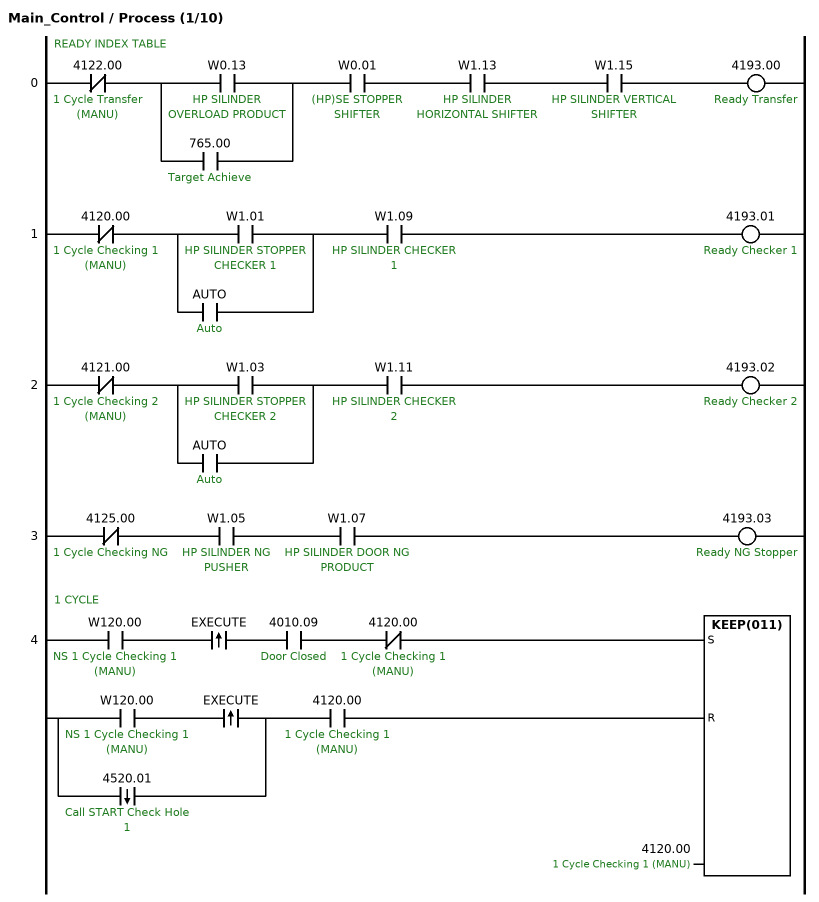
; [picture p24: Main_Control / Process, rungs 0-4]
; rung 0: READY INDEX TABLE
LDNOT 4122.00  ; 1 Cycle Transfer (MANU)
LD W0.13  ; HP SILINDER OVERLOAD PRODUCT
OR 765.00  ; Target Achieve
ANDLD
AND W0.01  ; (HP)SE STOPPER SHIFTER
AND W1.13  ; HP SILINDER HORIZONTAL SHIFTER
AND W1.15  ; HP SILINDER VERTICAL SHIFTER
OUT 4193.00  ; Ready Transfer
; rung 1
LDNOT 4120.00  ; 1 Cycle Checking 1 (MANU)
LD W1.01  ; HP SILINDER STOPPER CHECKER 1
OR AUTO  ; Auto
ANDLD
AND W1.09  ; HP SILINDER CHECKER 1
OUT 4193.01  ; Ready Checker 1
; rung 2
LDNOT 4121.00  ; 1 Cycle Checking 2 (MANU)
LD W1.03  ; HP SILINDER STOPPER CHECKER 2
OR AUTO  ; Auto
ANDLD
AND W1.11  ; HP SILINDER CHECKER 2
OUT 4193.02  ; Ready Checker 2
; rung 3
LDNOT 4125.00  ; 1 Cycle Checking NG
AND W1.05  ; HP SILINDER NG PUSHER
AND W1.07  ; HP SILINDER DOOR NG PRODUCT
OUT 4193.03  ; Ready NG Stopper
; rung 4: 1 CYCLE
LD W120.00  ; NS 1 Cycle Checking 1 (MANU)
@AND EXECUTE
AND 4010.09  ; Door Closed
ANDNOT 4120.00  ; 1 Cycle Checking 1 (MANU)
LD W120.00  ; NS 1 Cycle Checking 1 (MANU)
@AND EXECUTE
%OR 4520.01  ; Call START Check Hole 1
AND 4120.00  ; 1 Cycle Checking 1 (MANU)
KEEP(011) 4120.00  ; 1 Cycle Checking 1 (MANU)

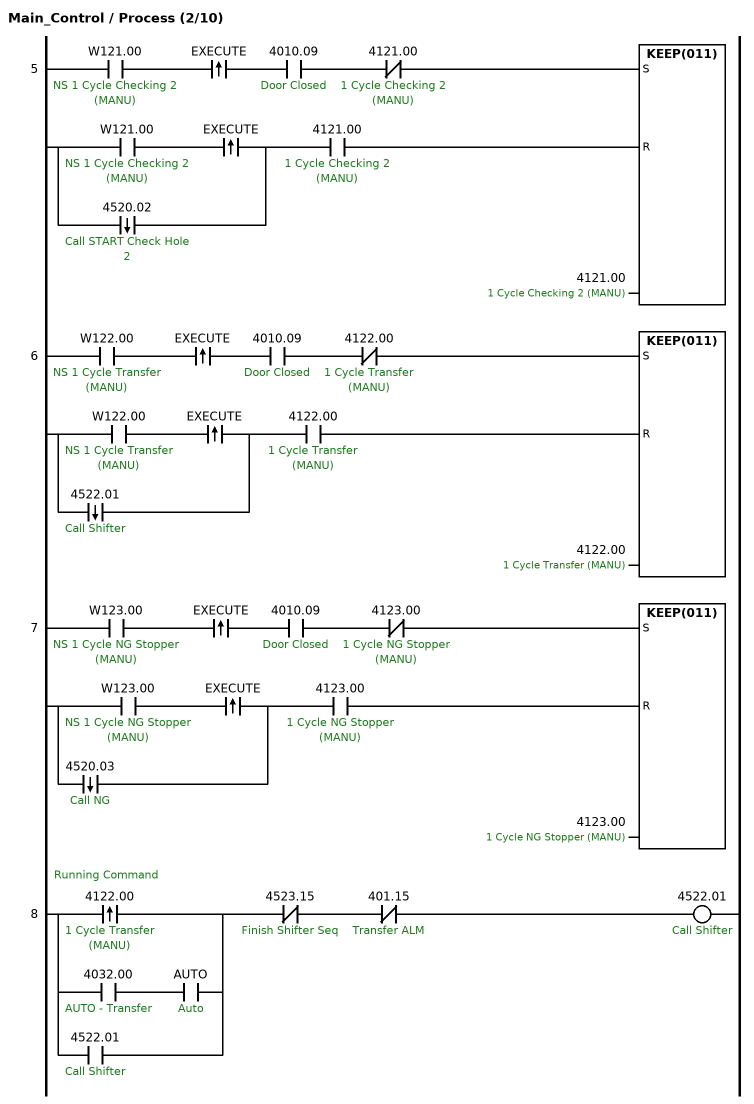
; rung 5
LD W121.00  ; NS 1 Cycle Checking 2 (MANU)
@AND EXECUTE
AND 4010.09  ; Door Closed
ANDNOT 4121.00  ; 1 Cycle Checking 2 (MANU)
LD W121.00  ; NS 1 Cycle Checking 2 (MANU)
@AND EXECUTE
%OR 4520.02  ; Call START Check Hole 2
AND 4121.00  ; 1 Cycle Checking 2 (MANU)
KEEP(011) 4121.00  ; 1 Cycle Checking 2 (MANU)
; rung 6
LD W122.00  ; NS 1 Cycle Transfer  (MANU)
@AND EXECUTE
AND 4010.09  ; Door Closed
ANDNOT 4122.00  ; 1 Cycle Transfer (MANU)
LD W122.00  ; NS 1 Cycle Transfer  (MANU)
@AND EXECUTE
%OR 4522.01  ; Call Shifter
AND 4122.00  ; 1 Cycle Transfer (MANU)
KEEP(011) 4122.00  ; 1 Cycle Transfer (MANU)
; rung 7
LD W123.00  ; NS 1 Cycle NG Stopper (MANU)
@AND EXECUTE
AND 4010.09  ; Door Closed
ANDNOT 4123.00  ; 1 Cycle NG Stopper (MANU)
LD W123.00  ; NS 1 Cycle NG Stopper (MANU)
@AND EXECUTE
%OR 4520.03  ; Call NG
AND 4123.00  ; 1 Cycle NG Stopper (MANU)
KEEP(011) 4123.00  ; 1 Cycle NG Stopper (MANU)
; rung 8: Running Command
@LD 4122.00  ; 1 Cycle Transfer (MANU)
LD 4032.00  ; AUTO - Transfer
AND AUTO  ; Auto
ORLD
OR 4522.01  ; Call Shifter
ANDNOT 4523.15  ; Finish Shifter Seq
ANDNOT 401.15  ; Transfer ALM
OUT 4522.01  ; Call Shifter

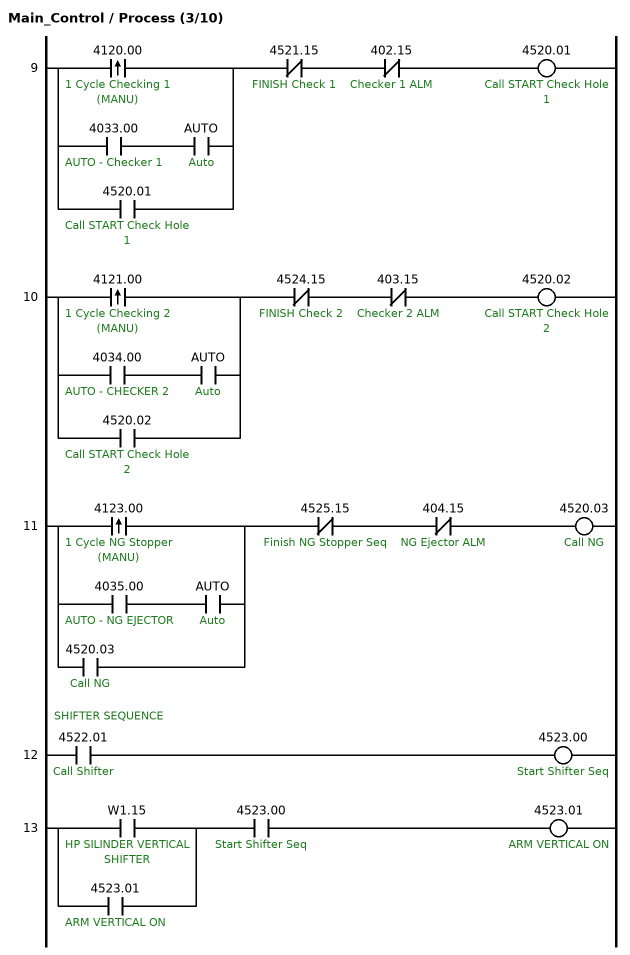
; rung 9
@LD 4120.00  ; 1 Cycle Checking 1 (MANU)
LD 4033.00  ; AUTO - Checker 1
AND AUTO  ; Auto
ORLD
OR 4520.01  ; Call START Check Hole 1
ANDNOT 4521.15  ; FINISH Check 1
ANDNOT 402.15  ; Checker 1 ALM
OUT 4520.01  ; Call START Check Hole 1
; rung 10
@LD 4121.00  ; 1 Cycle Checking 2 (MANU)
LD 4034.00  ; AUTO - CHECKER 2
AND AUTO  ; Auto
ORLD
OR 4520.02  ; Call START Check Hole 2
ANDNOT 4524.15  ; FINISH Check 2
ANDNOT 403.15  ; Checker 2 ALM
OUT 4520.02  ; Call START Check Hole 2
; rung 11
@LD 4123.00  ; 1 Cycle NG Stopper (MANU)
LD 4035.00  ; AUTO - NG EJECTOR
AND AUTO  ; Auto
ORLD
OR 4520.03  ; Call NG
ANDNOT 4525.15  ; Finish NG Stopper Seq
ANDNOT 404.15  ; NG Ejector ALM
OUT 4520.03  ; Call NG
; rung 12: SHIFTER SEQUENCE
LD 4522.01  ; Call Shifter
OUT 4523.00  ; Start Shifter Seq
; rung 13
LD W1.15  ; HP SILINDER VERTICAL SHIFTER
OR 4523.01  ; ARM VERTICAL ON
AND 4523.00  ; Start Shifter Seq
OUT 4523.01  ; ARM VERTICAL ON

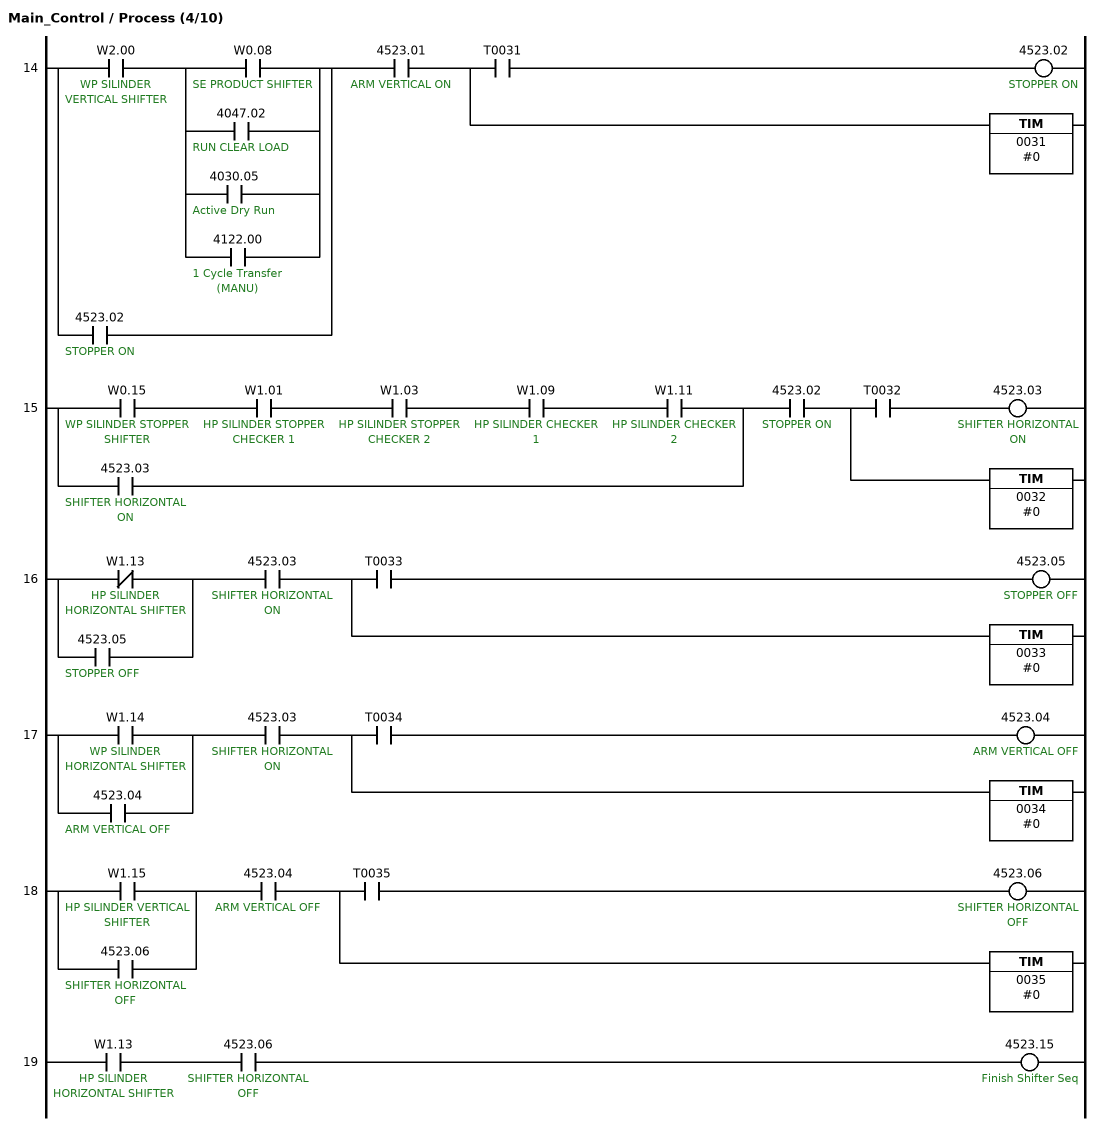
; rung 14
LD W2.00  ; WP SILINDER VERTICAL SHIFTER
LD W0.08  ; SE PRODUCT SHIFTER
OR 4047.02  ; RUN CLEAR LOAD
OR 4030.05  ; Active Dry Run
OR 4122.00  ; 1 Cycle Transfer (MANU)
ANDLD
OR 4523.02  ; STOPPER ON
AND 4523.01  ; ARM VERTICAL ON
OUT TR0
AND T0031
OUT 4523.02  ; STOPPER ON
LD TR0
TIM 0031 #0
; rung 15
LD W0.15  ; WP SILINDER STOPPER SHIFTER
AND W1.01  ; HP SILINDER STOPPER CHECKER 1
AND W1.03  ; HP SILINDER STOPPER CHECKER 2
AND W1.09  ; HP SILINDER CHECKER 1
AND W1.11  ; HP SILINDER CHECKER 2
OR 4523.03  ; SHIFTER HORIZONTAL ON
AND 4523.02  ; STOPPER ON
OUT TR0
AND T0032
OUT 4523.03  ; SHIFTER HORIZONTAL ON
LD TR0
TIM 0032 #0
; rung 16
LDNOT W1.13  ; HP SILINDER HORIZONTAL SHIFTER
OR 4523.05  ; STOPPER OFF
AND 4523.03  ; SHIFTER HORIZONTAL ON
OUT TR0
AND T0033
OUT 4523.05  ; STOPPER OFF
LD TR0
TIM 0033 #0
; rung 17
LD W1.14  ; WP SILINDER HORIZONTAL SHIFTER
OR 4523.04  ; ARM VERTICAL OFF
AND 4523.03  ; SHIFTER HORIZONTAL ON
OUT TR0
AND T0034
OUT 4523.04  ; ARM VERTICAL OFF
LD TR0
TIM 0034 #0
; rung 18
LD W1.15  ; HP SILINDER VERTICAL SHIFTER
OR 4523.06  ; SHIFTER HORIZONTAL OFF
AND 4523.04  ; ARM VERTICAL OFF
OUT TR0
AND T0035
OUT 4523.06  ; SHIFTER HORIZONTAL OFF
LD TR0
TIM 0035 #0
; rung 19
LD W1.13  ; HP SILINDER HORIZONTAL SHIFTER
AND 4523.06  ; SHIFTER HORIZONTAL OFF
OUT 4523.15  ; Finish Shifter Seq

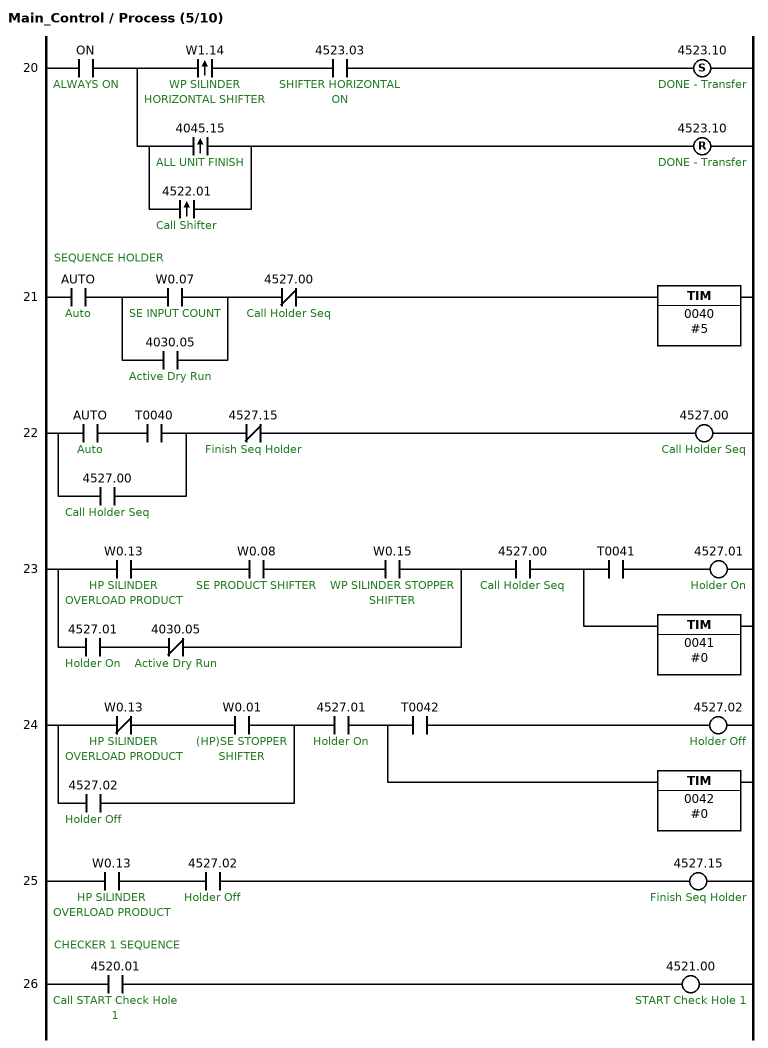
; rung 20
LD ON  ; ALWAYS ON
OUT TR0
@AND W1.14  ; WP SILINDER HORIZONTAL SHIFTER
AND 4523.03  ; SHIFTER HORIZONTAL ON
SET 4523.10  ; DONE - Transfer
LD TR0
@LD 4045.15  ; ALL UNIT FINISH
@OR 4522.01  ; Call Shifter
ANDLD
RSET 4523.10  ; DONE - Transfer
; rung 21: SEQUENCE HOLDER
LD AUTO  ; Auto
LD W0.07  ; SE INPUT COUNT
OR 4030.05  ; Active Dry Run
ANDLD
ANDNOT 4527.00  ; Call Holder Seq
TIM 0040 #5
; rung 22
LD AUTO  ; Auto
AND T0040
OR 4527.00  ; Call Holder Seq
ANDNOT 4527.15  ; Finish Seq Holder
OUT 4527.00  ; Call Holder Seq
; rung 23
LD W0.13  ; HP SILINDER OVERLOAD PRODUCT
AND W0.08  ; SE PRODUCT SHIFTER
AND W0.15  ; WP SILINDER STOPPER SHIFTER
LD 4527.01  ; Holder On
ANDNOT 4030.05  ; Active Dry Run
ORLD
AND 4527.00  ; Call Holder Seq
OUT TR0
AND T0041
OUT 4527.01  ; Holder On
LD TR0
TIM 0041 #0
; rung 24
LDNOT W0.13  ; HP SILINDER OVERLOAD PRODUCT
AND W0.01  ; (HP)SE STOPPER SHIFTER
OR 4527.02  ; Holder Off
AND 4527.01  ; Holder On
OUT TR0
AND T0042
OUT 4527.02  ; Holder Off
LD TR0
TIM 0042 #0
; rung 25
LD W0.13  ; HP SILINDER OVERLOAD PRODUCT
AND 4527.02  ; Holder Off
OUT 4527.15  ; Finish Seq Holder
; rung 26: CHECKER 1 SEQUENCE
LD 4520.01  ; Call START Check Hole 1
OUT 4521.00  ; START Check Hole 1

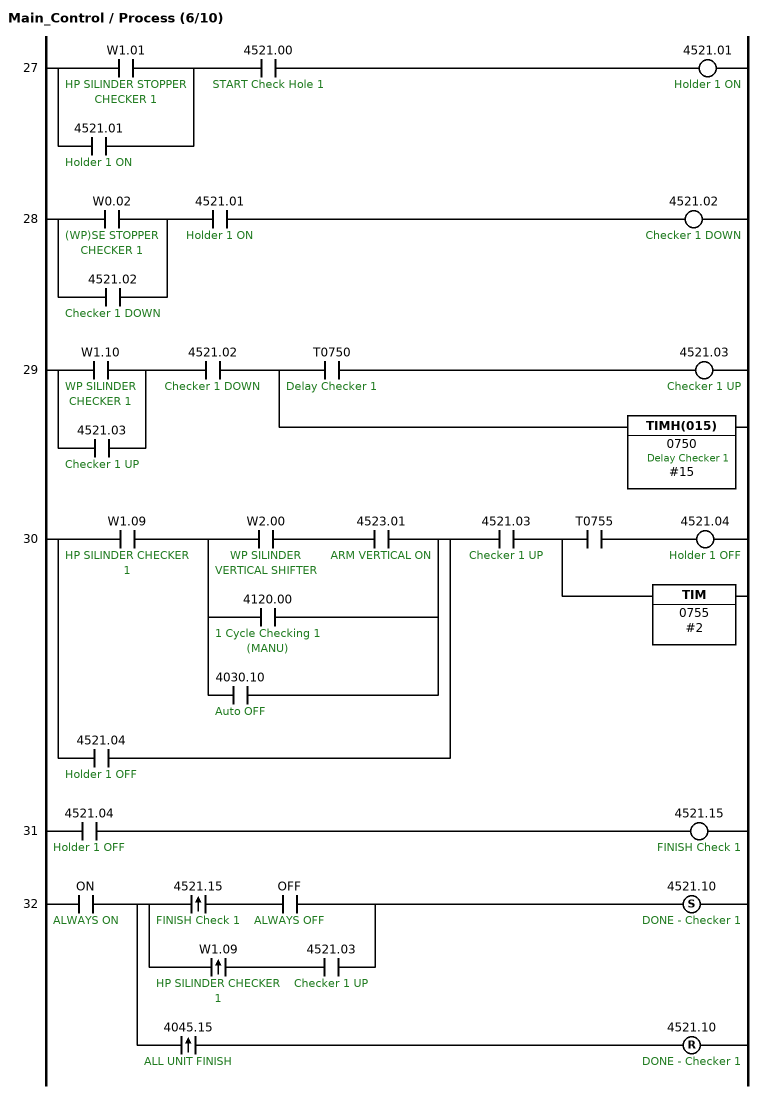
; rung 27
LD W1.01  ; HP SILINDER STOPPER CHECKER 1
OR 4521.01  ; Holder 1 ON
AND 4521.00  ; START Check Hole 1
OUT 4521.01  ; Holder 1 ON
; rung 28
LD W0.02  ; (WP)SE STOPPER CHECKER 1
OR 4521.02  ; Checker 1 DOWN
AND 4521.01  ; Holder 1 ON
OUT 4521.02  ; Checker 1 DOWN
; rung 29
LD W1.10  ; WP SILINDER CHECKER 1
OR 4521.03  ; Checker 1 UP
AND 4521.02  ; Checker 1 DOWN
OUT TR0
AND T0750  ; Delay Checker 1
OUT 4521.03  ; Checker 1 UP
LD TR0
TIMH(015) 0750 #15  ; Delay Checker 1
; rung 30
LD W1.09  ; HP SILINDER CHECKER 1
LD W2.00  ; WP SILINDER VERTICAL SHIFTER
AND 4523.01  ; ARM VERTICAL ON
OR 4120.00  ; 1 Cycle Checking 1 (MANU)
OR 4030.10  ; Auto OFF
ANDLD
OR 4521.04  ; Holder 1 OFF
AND 4521.03  ; Checker 1 UP
OUT TR0
AND T0755
OUT 4521.04  ; Holder 1 OFF
LD TR0
TIM 0755 #2
; rung 31
LD 4521.04  ; Holder 1 OFF
OUT 4521.15  ; FINISH Check 1
; rung 32
LD ON  ; ALWAYS ON
OUT TR0
@LD 4521.15  ; FINISH Check 1
AND OFF  ; ALWAYS OFF
@LD W1.09  ; HP SILINDER CHECKER 1
AND 4521.03  ; Checker 1 UP
ORLD
ANDLD
SET 4521.10  ; DONE - Checker 1
LD TR0
@AND 4045.15  ; ALL UNIT FINISH
RSET 4521.10  ; DONE - Checker 1

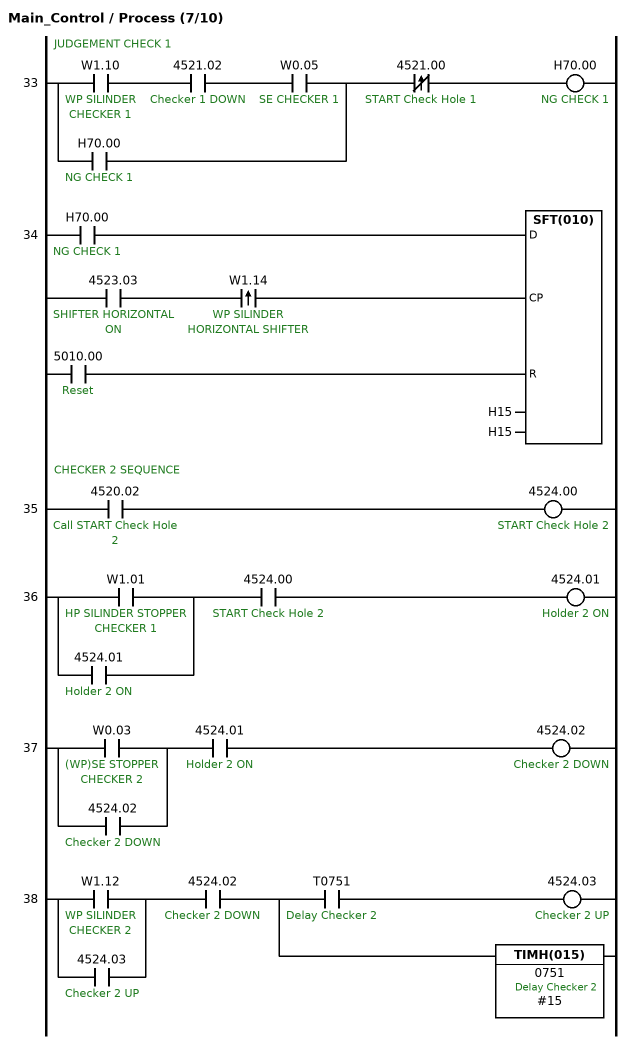
; rung 33: JUDGEMENT CHECK 1
LD W1.10  ; WP SILINDER CHECKER 1
AND 4521.02  ; Checker 1 DOWN
AND W0.05  ; SE CHECKER 1
OR H70.00  ; NG CHECK 1
@ANDNOT 4521.00  ; START Check Hole 1
OUT H70.00  ; NG CHECK 1
; rung 34
LD H70.00  ; NG CHECK 1
LD 4523.03  ; SHIFTER HORIZONTAL ON
@AND W1.14  ; WP SILINDER HORIZONTAL SHIFTER
LD 5010.00  ; Reset
SFT(010) H15 H15
; rung 35: CHECKER 2 SEQUENCE
LD 4520.02  ; Call START Check Hole 2
OUT 4524.00  ; START Check Hole 2
; rung 36
LD W1.01  ; HP SILINDER STOPPER CHECKER 1
OR 4524.01  ; Holder 2 ON
AND 4524.00  ; START Check Hole 2
OUT 4524.01  ; Holder 2 ON
; rung 37
LD W0.03  ; (WP)SE STOPPER CHECKER 2
OR 4524.02  ; Checker 2 DOWN
AND 4524.01  ; Holder 2 ON
OUT 4524.02  ; Checker 2 DOWN
; rung 38
LD W1.12  ; WP SILINDER CHECKER 2
OR 4524.03  ; Checker 2 UP
AND 4524.02  ; Checker 2 DOWN
OUT TR0
AND T0751  ; Delay Checker 2
OUT 4524.03  ; Checker 2 UP
LD TR0
TIMH(015) 0751 #15  ; Delay Checker 2

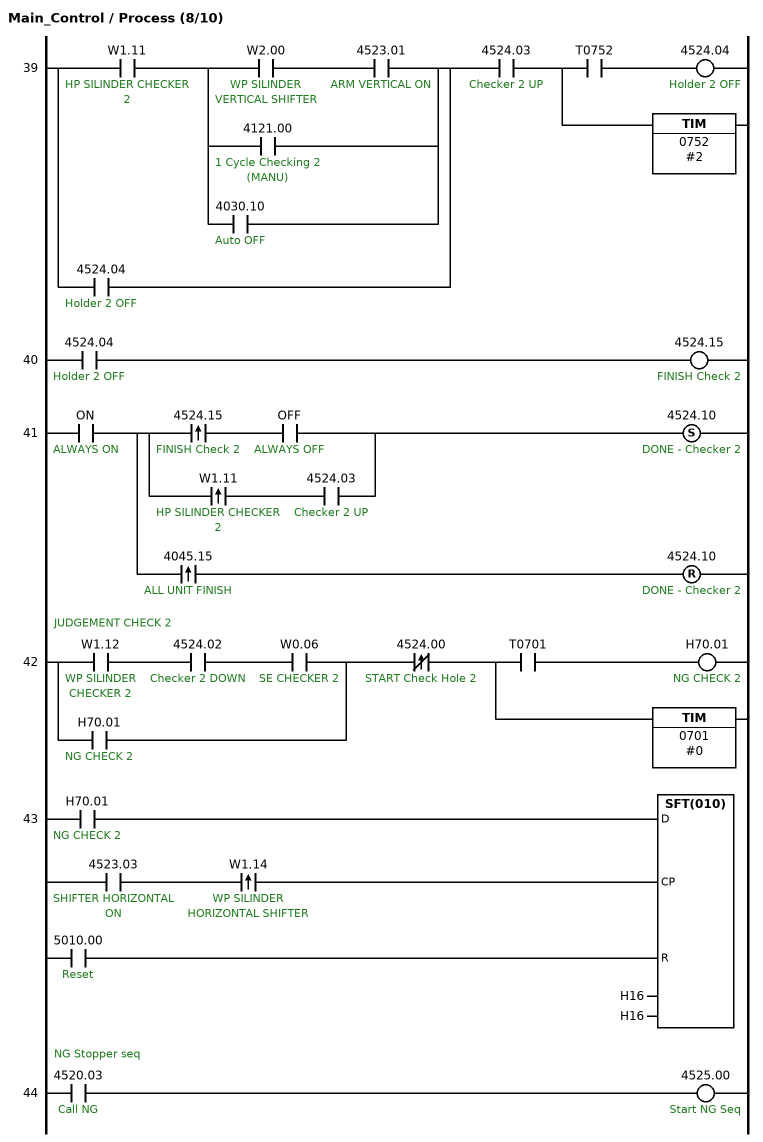
; rung 39
LD W1.11  ; HP SILINDER CHECKER 2
LD W2.00  ; WP SILINDER VERTICAL SHIFTER
AND 4523.01  ; ARM VERTICAL ON
OR 4121.00  ; 1 Cycle Checking 2 (MANU)
OR 4030.10  ; Auto OFF
ANDLD
OR 4524.04  ; Holder 2 OFF
AND 4524.03  ; Checker 2 UP
OUT TR0
AND T0752
OUT 4524.04  ; Holder 2 OFF
LD TR0
TIM 0752 #2
; rung 40
LD 4524.04  ; Holder 2 OFF
OUT 4524.15  ; FINISH Check 2
; rung 41
LD ON  ; ALWAYS ON
OUT TR0
@LD 4524.15  ; FINISH Check 2
AND OFF  ; ALWAYS OFF
@LD W1.11  ; HP SILINDER CHECKER 2
AND 4524.03  ; Checker 2 UP
ORLD
ANDLD
SET 4524.10  ; DONE - Checker 2
LD TR0
@AND 4045.15  ; ALL UNIT FINISH
RSET 4524.10  ; DONE - Checker 2
; rung 42: JUDGEMENT CHECK 2
LD W1.12  ; WP SILINDER CHECKER 2
AND 4524.02  ; Checker 2 DOWN
AND W0.06  ; SE CHECKER 2
OR H70.01  ; NG CHECK 2
@ANDNOT 4524.00  ; START Check Hole 2
OUT TR0
AND T0701
OUT H70.01  ; NG CHECK 2
LD TR0
TIM 0701 #0
; rung 43
LD H70.01  ; NG CHECK 2
LD 4523.03  ; SHIFTER HORIZONTAL ON
@AND W1.14  ; WP SILINDER HORIZONTAL SHIFTER
LD 5010.00  ; Reset
SFT(010) H16 H16
; rung 44: NG Stopper seq
LD 4520.03  ; Call NG
OUT 4525.00  ; Start NG Seq

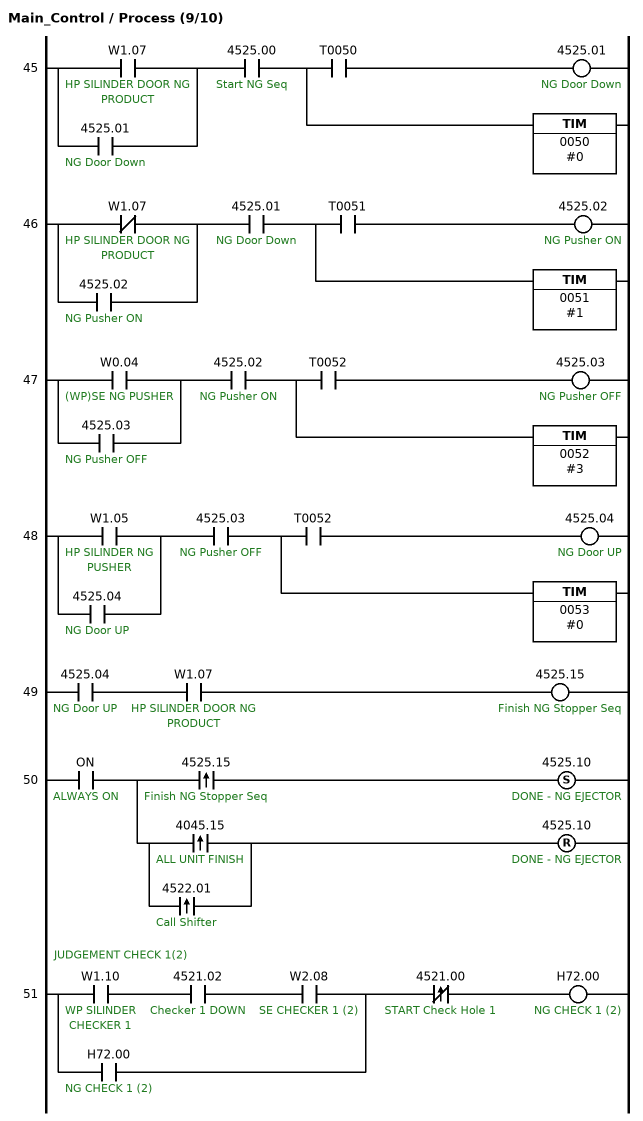
; rung 45
LD W1.07  ; HP SILINDER DOOR NG PRODUCT
OR 4525.01  ; NG Door Down
AND 4525.00  ; Start NG Seq
OUT TR0
AND T0050
OUT 4525.01  ; NG Door Down
LD TR0
TIM 0050 #0
; rung 46
LDNOT W1.07  ; HP SILINDER DOOR NG PRODUCT
OR 4525.02  ; NG Pusher ON
AND 4525.01  ; NG Door Down
OUT TR0
AND T0051
OUT 4525.02  ; NG Pusher ON
LD TR0
TIM 0051 #1
; rung 47
LD W0.04  ; (WP)SE NG PUSHER
OR 4525.03  ; NG Pusher OFF
AND 4525.02  ; NG Pusher ON
OUT TR0
AND T0052
OUT 4525.03  ; NG Pusher OFF
LD TR0
TIM 0052 #3
; rung 48
LD W1.05  ; HP SILINDER NG PUSHER
OR 4525.04  ; NG Door UP
AND 4525.03  ; NG Pusher OFF
OUT TR0
AND T0052
OUT 4525.04  ; NG Door UP
LD TR0
TIM 0053 #0
; rung 49
LD 4525.04  ; NG Door UP
AND W1.07  ; HP SILINDER DOOR NG PRODUCT
OUT 4525.15  ; Finish NG Stopper Seq
; rung 50
LD ON  ; ALWAYS ON
OUT TR0
@AND 4525.15  ; Finish NG Stopper Seq
SET 4525.10  ; DONE - NG EJECTOR
LD TR0
@LD 4045.15  ; ALL UNIT FINISH
@OR 4522.01  ; Call Shifter
ANDLD
RSET 4525.10  ; DONE - NG EJECTOR
; rung 51: JUDGEMENT CHECK 1(2)
LD W1.10  ; WP SILINDER CHECKER 1
AND 4521.02  ; Checker 1 DOWN
AND W2.08  ; SE CHECKER 1 (2)
OR H72.00  ; NG CHECK 1 (2)
@ANDNOT 4521.00  ; START Check Hole 1
OUT H72.00  ; NG CHECK 1 (2)

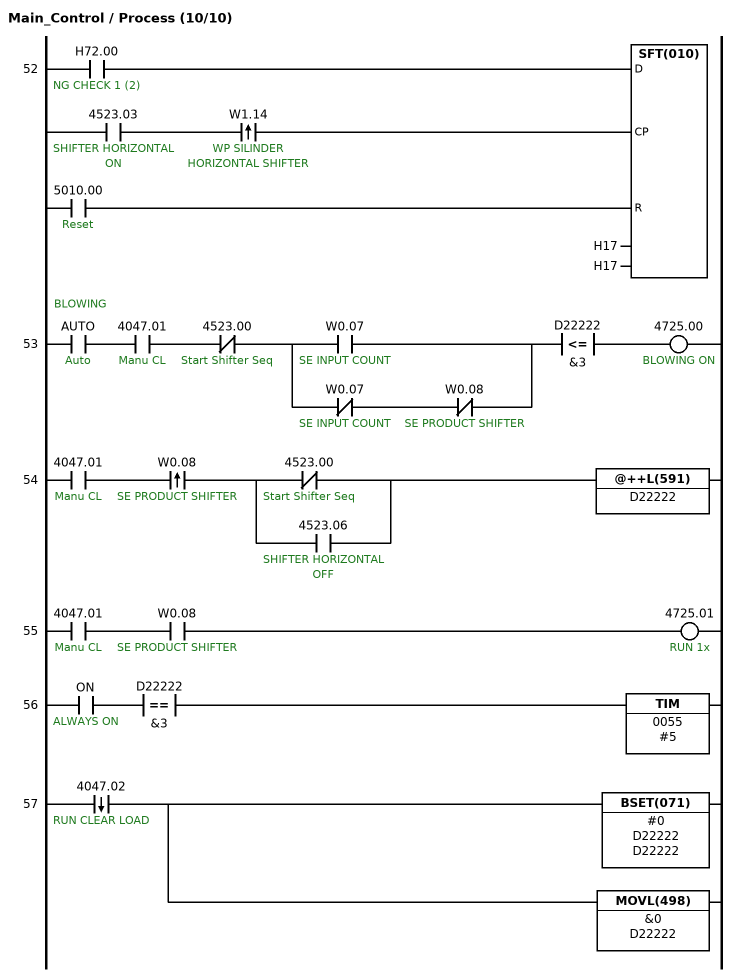
; rung 52
LD H72.00  ; NG CHECK 1 (2)
LD 4523.03  ; SHIFTER HORIZONTAL ON
@AND W1.14  ; WP SILINDER HORIZONTAL SHIFTER
LD 5010.00  ; Reset
SFT(010) H17 H17
; rung 53: BLOWING
LD AUTO  ; Auto
AND 4047.01  ; Manu CL
ANDNOT 4523.00  ; Start Shifter Seq
LD W0.07  ; SE INPUT COUNT
LDNOT W0.07  ; SE INPUT COUNT
ANDNOT W0.08  ; SE PRODUCT SHIFTER
ORLD
ANDLD
AND<=(315) D22222 &3
OUT 4725.00  ; BLOWING ON
; rung 54
LD 4047.01  ; Manu CL
@AND W0.08  ; SE PRODUCT SHIFTER
LDNOT 4523.00  ; Start Shifter Seq
OR 4523.06  ; SHIFTER HORIZONTAL OFF
ANDLD
@++L(591) D22222
; rung 55
LD 4047.01  ; Manu CL
AND W0.08  ; SE PRODUCT SHIFTER
OUT 4725.01  ; RUN 1x
; rung 56
LD ON  ; ALWAYS ON
AND=(300) D22222 &3
TIM 0055 #5
; rung 57
%LD 4047.02  ; RUN CLEAR LOAD
BSET(071) #0 D22222 D22222
MOVL(498) &0 D22222

### Section All_Unit_Status

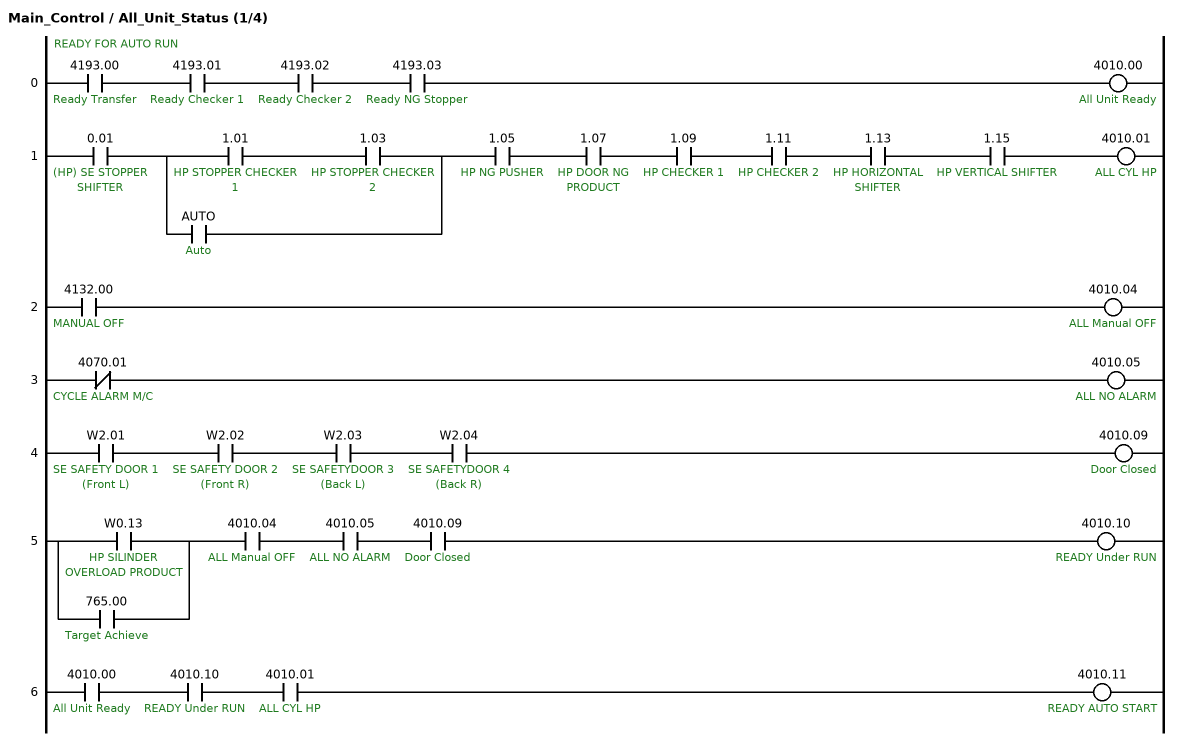
; rung 0: READY FOR AUTO RUN
LD 4193.00  ; Ready Transfer
AND 4193.01  ; Ready Checker 1
AND 4193.02  ; Ready Checker 2
AND 4193.03  ; Ready NG Stopper
OUT 4010.00  ; All Unit Ready
; rung 1
LD 0.01  ; (HP) SE STOPPER SHIFTER
LD 1.01  ; HP STOPPER CHECKER 1
AND 1.03  ; HP STOPPER CHECKER 2
OR AUTO  ; Auto
ANDLD
AND 1.05  ; HP NG PUSHER
AND 1.07  ; HP DOOR NG PRODUCT
AND 1.09  ; HP CHECKER 1
AND 1.11  ; HP CHECKER 2
AND 1.13  ; HP HORIZONTAL SHIFTER
AND 1.15  ; HP VERTICAL SHIFTER
OUT 4010.01  ; ALL CYL HP
; rung 2
LD 4132.00  ; MANUAL OFF
OUT 4010.04  ; ALL Manual OFF
; rung 3
LDNOT 4070.01  ; CYCLE ALARM M/C
OUT 4010.05  ; ALL NO ALARM
; rung 4
LD W2.01  ; SE SAFETY DOOR 1 (Front L)
AND W2.02  ; SE SAFETY DOOR 2 (Front R)
AND W2.03  ; SE SAFETYDOOR 3 (Back L)
AND W2.04  ; SE SAFETYDOOR 4 (Back R)
OUT 4010.09  ; Door Closed
; rung 5
LD W0.13  ; HP SILINDER OVERLOAD PRODUCT
OR 765.00  ; Target Achieve
AND 4010.04  ; ALL Manual OFF
AND 4010.05  ; ALL NO ALARM
AND 4010.09  ; Door Closed
OUT 4010.10  ; READY Under RUN
; rung 6
LD 4010.00  ; All Unit Ready
AND 4010.10  ; READY Under RUN
AND 4010.01  ; ALL CYL HP
OUT 4010.11  ; READY AUTO START

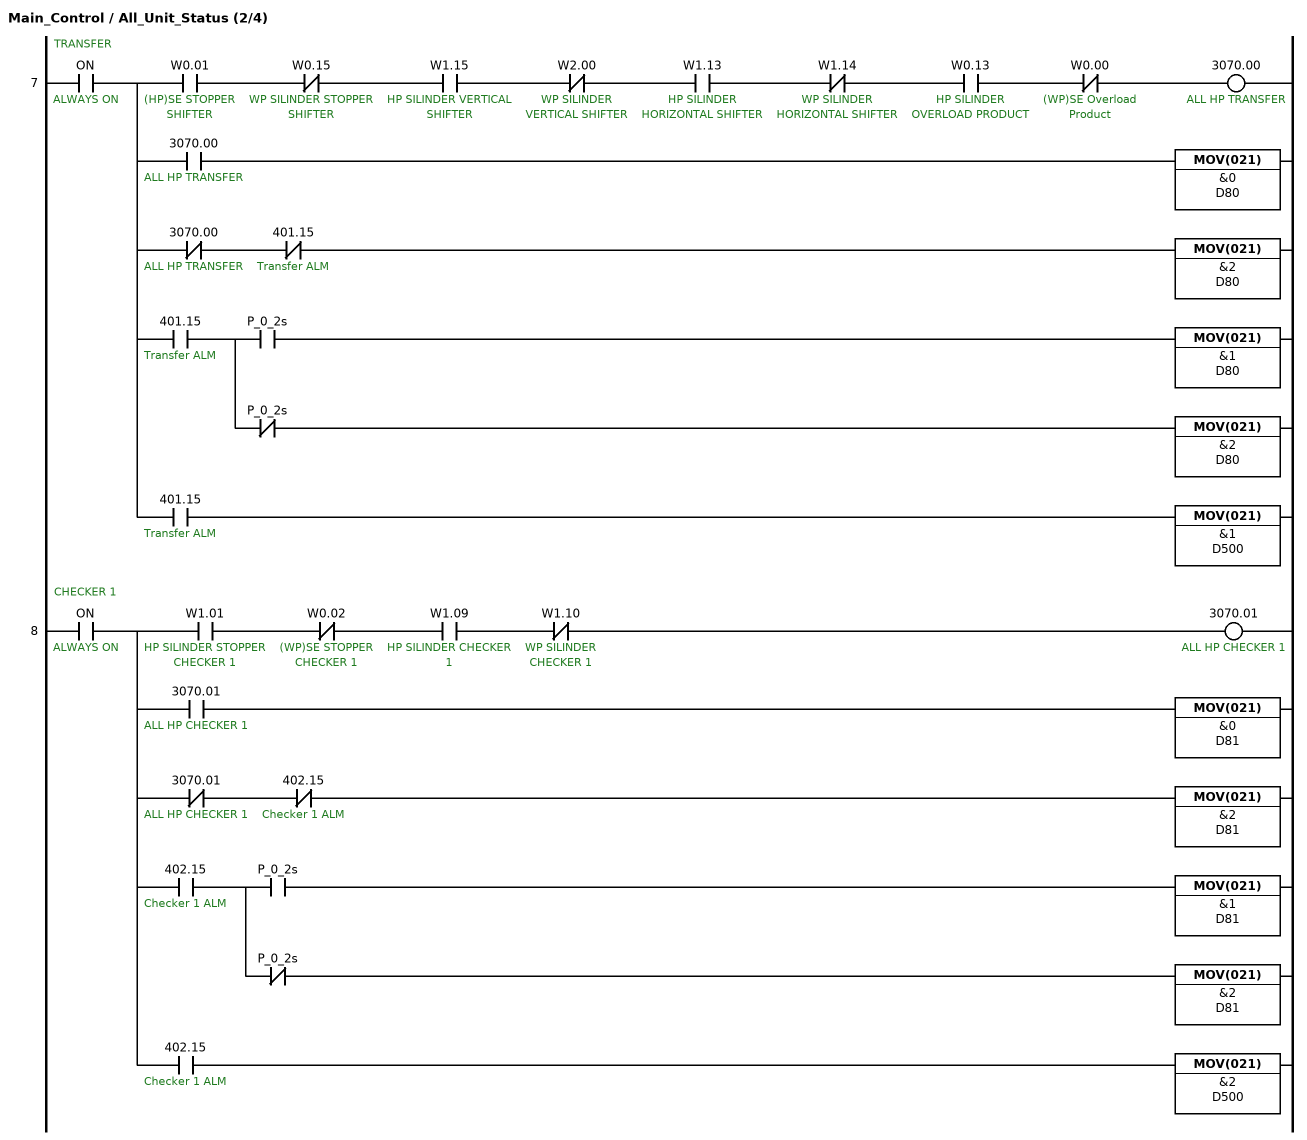
; rung 7: TRANSFER
LD ON  ; ALWAYS ON
OUT TR0
AND W0.01  ; (HP)SE STOPPER SHIFTER
ANDNOT W0.15  ; WP SILINDER STOPPER SHIFTER
AND W1.15  ; HP SILINDER VERTICAL SHIFTER
ANDNOT W2.00  ; WP SILINDER VERTICAL SHIFTER
AND W1.13  ; HP SILINDER HORIZONTAL SHIFTER
ANDNOT W1.14  ; WP SILINDER HORIZONTAL SHIFTER
AND W0.13  ; HP SILINDER OVERLOAD PRODUCT
ANDNOT W0.00  ; (WP)SE Overload Product
OUT 3070.00  ; ALL HP TRANSFER
LD TR0
AND 3070.00  ; ALL HP TRANSFER
MOV(021) &0 D80
LD TR0
ANDNOT 3070.00  ; ALL HP TRANSFER
ANDNOT 401.15  ; Transfer ALM
MOV(021) &2 D80
LD TR0
AND 401.15  ; Transfer ALM
OUT TR1
AND P_0_2s
MOV(021) &1 D80
LD TR1
ANDNOT P_0_2s
MOV(021) &2 D80
LD TR0
AND 401.15  ; Transfer ALM
MOV(021) &1 D500
; rung 8: CHECKER 1
LD ON  ; ALWAYS ON
OUT TR0
AND W1.01  ; HP SILINDER STOPPER CHECKER 1
ANDNOT W0.02  ; (WP)SE STOPPER CHECKER 1
AND W1.09  ; HP SILINDER CHECKER 1
ANDNOT W1.10  ; WP SILINDER CHECKER 1
OUT 3070.01  ; ALL HP CHECKER 1
LD TR0
AND 3070.01  ; ALL HP CHECKER 1
MOV(021) &0 D81
LD TR0
ANDNOT 3070.01  ; ALL HP CHECKER 1
ANDNOT 402.15  ; Checker 1 ALM
MOV(021) &2 D81
LD TR0
AND 402.15  ; Checker 1 ALM
OUT TR1
AND P_0_2s
MOV(021) &1 D81
LD TR1
ANDNOT P_0_2s
MOV(021) &2 D81
LD TR0
AND 402.15  ; Checker 1 ALM
MOV(021) &2 D500

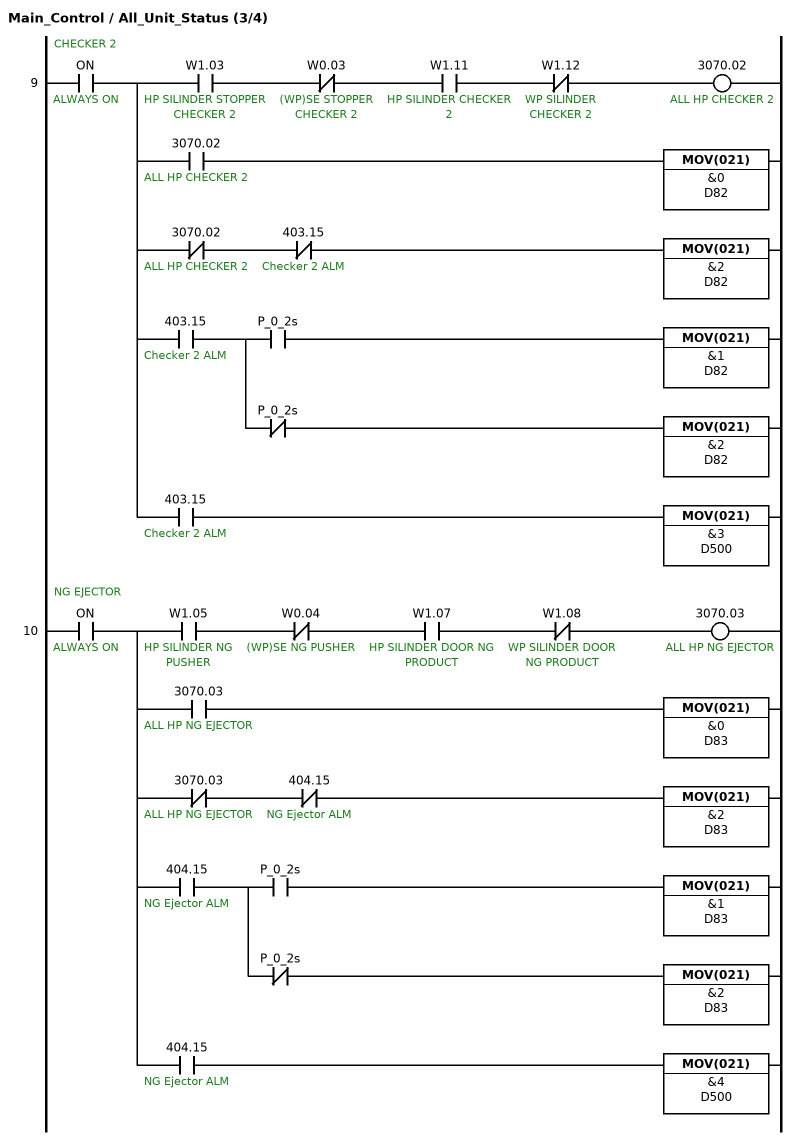
; rung 9: CHECKER 2
LD ON  ; ALWAYS ON
OUT TR0
AND W1.03  ; HP SILINDER STOPPER CHECKER 2
ANDNOT W0.03  ; (WP)SE STOPPER CHECKER 2
AND W1.11  ; HP SILINDER CHECKER 2
ANDNOT W1.12  ; WP SILINDER CHECKER 2
OUT 3070.02  ; ALL HP CHECKER 2
LD TR0
AND 3070.02  ; ALL HP CHECKER 2
MOV(021) &0 D82
LD TR0
ANDNOT 3070.02  ; ALL HP CHECKER 2
ANDNOT 403.15  ; Checker 2 ALM
MOV(021) &2 D82
LD TR0
AND 403.15  ; Checker 2 ALM
OUT TR1
AND P_0_2s
MOV(021) &1 D82
LD TR1
ANDNOT P_0_2s
MOV(021) &2 D82
LD TR0
AND 403.15  ; Checker 2 ALM
MOV(021) &3 D500
; rung 10: NG EJECTOR
LD ON  ; ALWAYS ON
OUT TR0
AND W1.05  ; HP SILINDER NG PUSHER
ANDNOT W0.04  ; (WP)SE NG PUSHER
AND W1.07  ; HP SILINDER DOOR NG PRODUCT
ANDNOT W1.08  ; WP SILINDER DOOR NG PRODUCT
OUT 3070.03  ; ALL HP NG EJECTOR
LD TR0
AND 3070.03  ; ALL HP NG EJECTOR
MOV(021) &0 D83
LD TR0
ANDNOT 3070.03  ; ALL HP NG EJECTOR
ANDNOT 404.15  ; NG Ejector ALM
MOV(021) &2 D83
LD TR0
AND 404.15  ; NG Ejector ALM
OUT TR1
AND P_0_2s
MOV(021) &1 D83
LD TR1
ANDNOT P_0_2s
MOV(021) &2 D83
LD TR0
AND 404.15  ; NG Ejector ALM
MOV(021) &4 D500

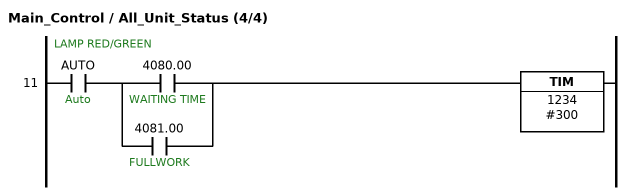
; rung 11: LAMP RED/GREEN
LD AUTO  ; Auto
LD 4080.00  ; WAITING TIME
OR 4081.00  ; FULLWORK
ANDLD
TIM 1234 #300
; rung 12: ADDITIONAL VISION -VER2-

### Section Unit_Setting

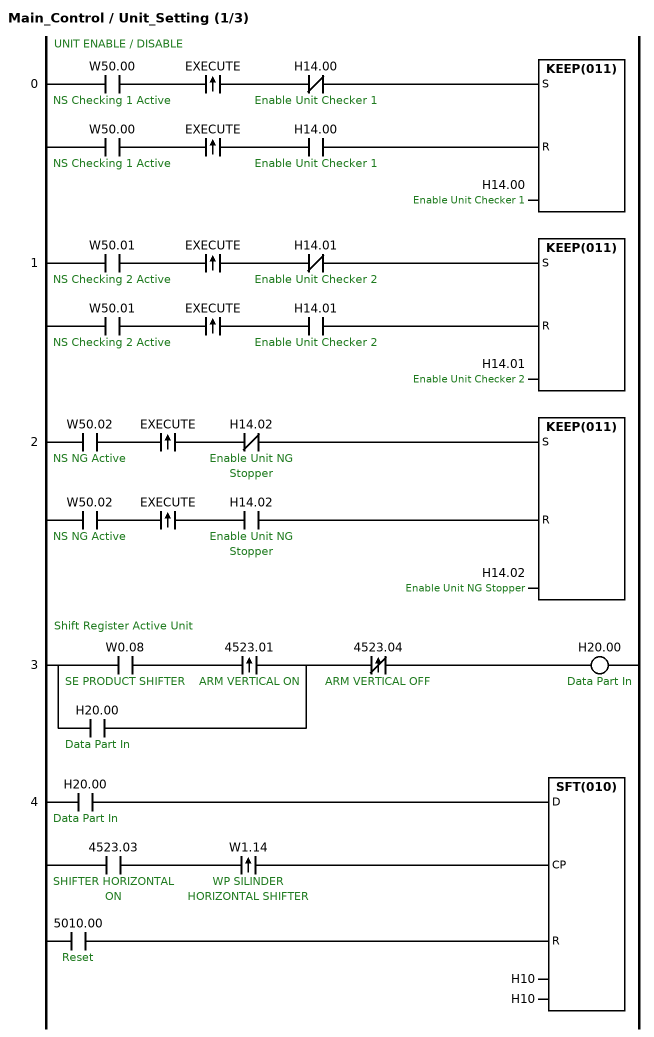
; rung 0: UNIT ENABLE / DISABLE
LD W50.00  ; NS Checking 1 Active
@AND EXECUTE
ANDNOT H14.00  ; Enable Unit Checker 1
LD W50.00  ; NS Checking 1 Active
@AND EXECUTE
AND H14.00  ; Enable Unit Checker 1
KEEP(011) H14.00  ; Enable Unit Checker 1
; rung 1
LD W50.01  ; NS Checking 2 Active
@AND EXECUTE
ANDNOT H14.01  ; Enable Unit Checker 2
LD W50.01  ; NS Checking 2 Active
@AND EXECUTE
AND H14.01  ; Enable Unit Checker 2
KEEP(011) H14.01  ; Enable Unit Checker 2
; rung 2
LD W50.02  ; NS NG Active
@AND EXECUTE
ANDNOT H14.02  ; Enable Unit NG Stopper
LD W50.02  ; NS NG Active
@AND EXECUTE
AND H14.02  ; Enable Unit NG Stopper
KEEP(011) H14.02  ; Enable Unit NG Stopper
; rung 3: Shift Register Active Unit
LD W0.08  ; SE PRODUCT SHIFTER
@AND 4523.01  ; ARM VERTICAL ON
OR H20.00  ; Data Part In
@ANDNOT 4523.04  ; ARM VERTICAL OFF
OUT H20.00  ; Data Part In
; rung 4
LD H20.00  ; Data Part In
LD 4523.03  ; SHIFTER HORIZONTAL ON
@AND W1.14  ; WP SILINDER HORIZONTAL SHIFTER
LD 5010.00  ; Reset
SFT(010) H10 H10

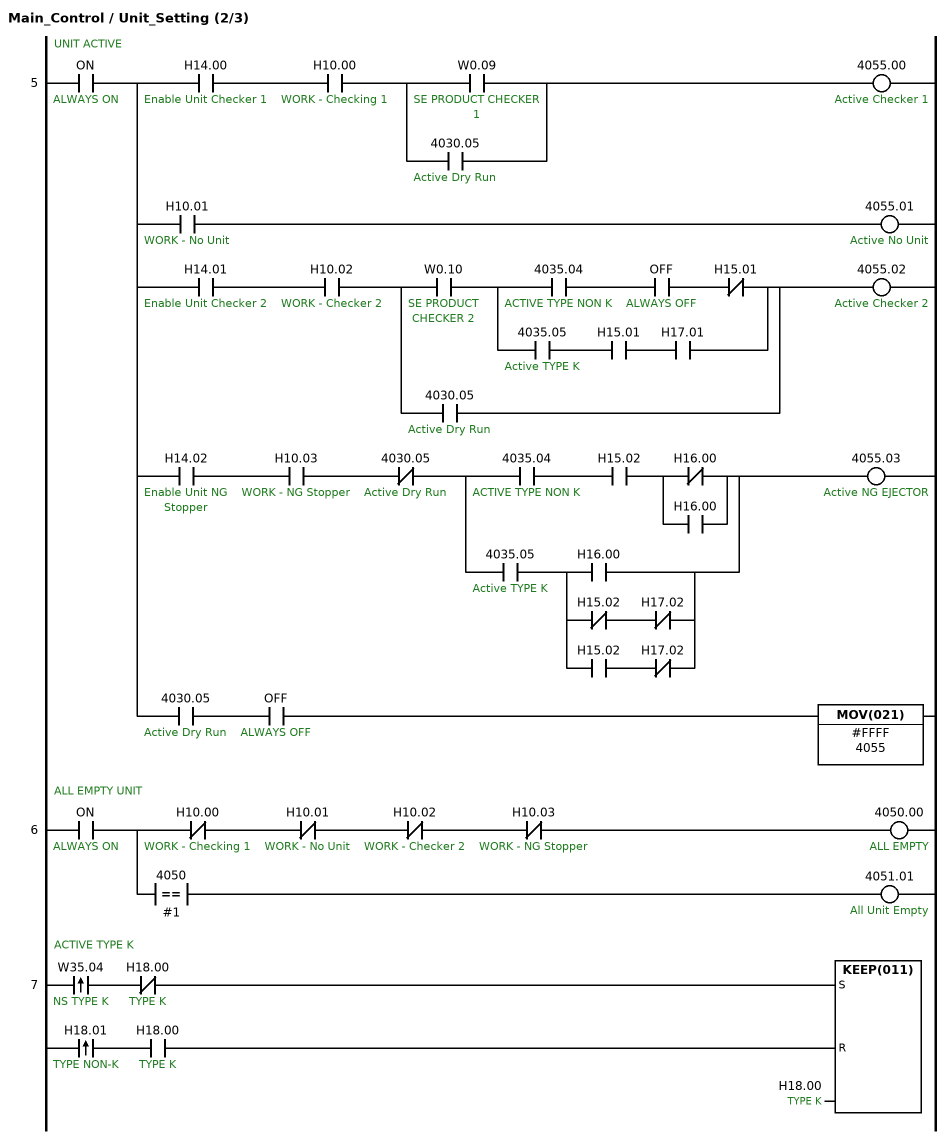
; rung 5: UNIT ACTIVE
LD ON  ; ALWAYS ON
OUT TR0
AND H14.00  ; Enable Unit Checker 1
AND H10.00  ; WORK - Checking 1
LD W0.09  ; SE PRODUCT CHECKER 1
OR 4030.05  ; Active Dry Run
ANDLD
OUT 4055.00  ; Active Checker 1
LD TR0
AND H10.01  ; WORK - No Unit
OUT 4055.01  ; Active No Unit
LD TR0
AND H14.01  ; Enable Unit Checker 2
AND H10.02  ; WORK - Checker 2
LD W0.10  ; SE PRODUCT  CHECKER 2
LD 4035.04  ; ACTIVE TYPE NON K
AND OFF  ; ALWAYS OFF
ANDNOT H15.01
LD 4035.05  ; Active TYPE K
AND H15.01
AND H17.01
ORLD
ANDLD
OR 4030.05  ; Active Dry Run
ANDLD
OUT 4055.02  ; Active Checker 2
LD TR0
AND H14.02  ; Enable Unit NG Stopper
AND H10.03  ; WORK - NG Stopper
ANDNOT 4030.05  ; Active Dry Run
LD 4035.04  ; ACTIVE TYPE NON K
AND H15.02
LDNOT H16.00
OR H16.00
ANDLD
LD 4035.05  ; Active TYPE K
LD H16.00
LDNOT H15.02
ANDNOT H17.02
ORLD
LD H15.02
ANDNOT H17.02
ORLD
ANDLD
ORLD
ANDLD
OUT 4055.03  ; Active NG EJECTOR
LD TR0
AND 4030.05  ; Active Dry Run
AND OFF  ; ALWAYS OFF
MOV(021) #FFFF 4055
; rung 6: ALL EMPTY UNIT
LD ON  ; ALWAYS ON
OUT TR0
ANDNOT H10.00  ; WORK - Checking 1
ANDNOT H10.01  ; WORK - No Unit
ANDNOT H10.02  ; WORK - Checker 2
ANDNOT H10.03  ; WORK - NG Stopper
OUT 4050.00  ; ALL EMPTY
LD TR0
AND=(300) 4050 #1
OUT 4051.01  ; All Unit Empty
; rung 7: ACTIVE TYPE K
@LD W35.04  ; NS TYPE K
ANDNOT H18.00  ; TYPE K
@LD H18.01  ; TYPE NON-K
AND H18.00  ; TYPE K
KEEP(011) H18.00  ; TYPE K

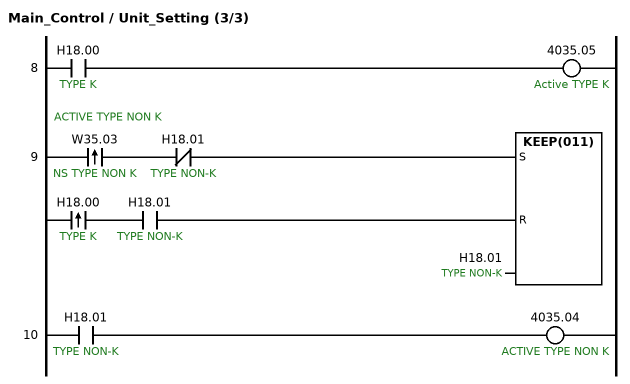
; rung 8
LD H18.00  ; TYPE K
OUT 4035.05  ; Active TYPE K
; rung 9: ACTIVE TYPE NON K
@LD W35.03  ; NS TYPE NON K
ANDNOT H18.01  ; TYPE NON-K
@LD H18.00  ; TYPE K
AND H18.01  ; TYPE NON-K
KEEP(011) H18.01  ; TYPE NON-K
; rung 10
LD H18.01  ; TYPE NON-K
OUT 4035.04  ; ACTIVE TYPE NON K

### Section PT_Control

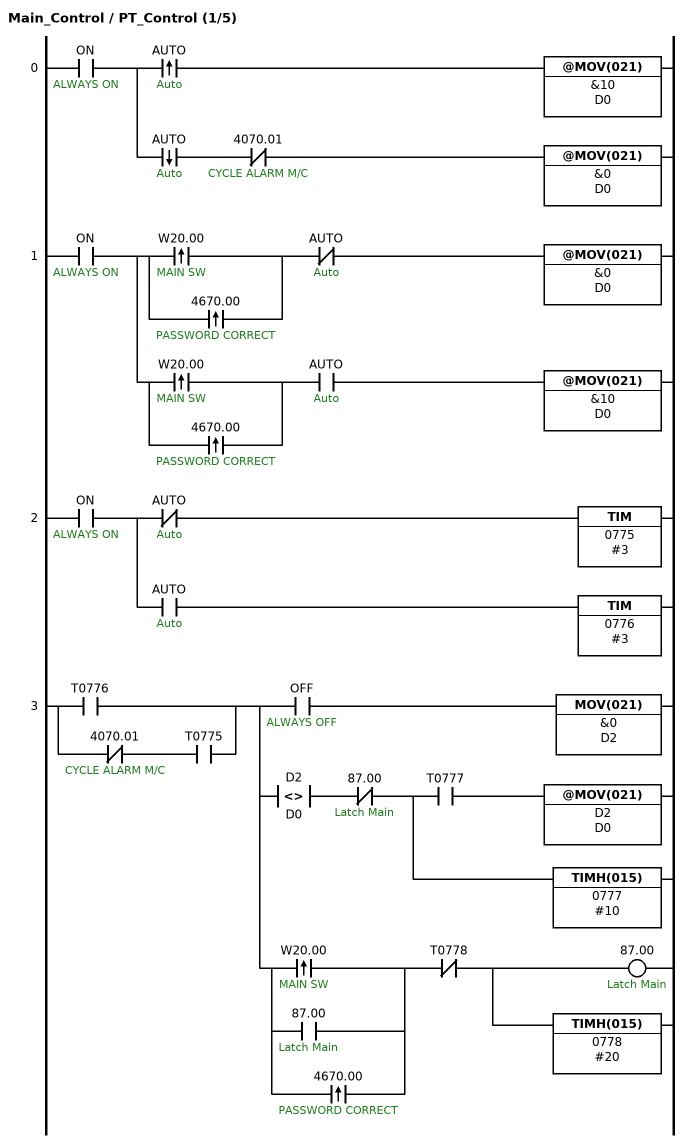
; rung 0
LD ON  ; ALWAYS ON
OUT TR0
@AND AUTO  ; Auto
@MOV(021) &10 D0
LD TR0
%AND AUTO  ; Auto
ANDNOT 4070.01  ; CYCLE ALARM M/C
@MOV(021) &0 D0
; rung 1
LD ON  ; ALWAYS ON
OUT TR0
@LD W20.00  ; MAIN SW
@OR 4670.00  ; PASSWORD CORRECT
ANDLD
ANDNOT AUTO  ; Auto
@MOV(021) &0 D0
LD TR0
@LD W20.00  ; MAIN SW
@OR 4670.00  ; PASSWORD CORRECT
ANDLD
AND AUTO  ; Auto
@MOV(021) &10 D0
; rung 2
LD ON  ; ALWAYS ON
OUT TR0
ANDNOT AUTO  ; Auto
TIM 0775 #3
LD TR0
AND AUTO  ; Auto
TIM 0776 #3
; rung 3
LD T0776
LDNOT 4070.01  ; CYCLE ALARM M/C
AND T0775
ORLD
OUT TR0
AND OFF  ; ALWAYS OFF
MOV(021) &0 D2
LD TR0
AND<>(305) D2 D0
ANDNOT 87.00  ; Latch Main
OUT TR1
AND T0777
@MOV(021) D2 D0
LD TR1
TIMH(015) 0777 #10
LD TR0
@LD W20.00  ; MAIN SW
OR 87.00  ; Latch Main
@OR 4670.00  ; PASSWORD CORRECT
ANDLD
ANDNOT T0778
OUT 87.00  ; Latch Main
TIMH(015) 0778 #20

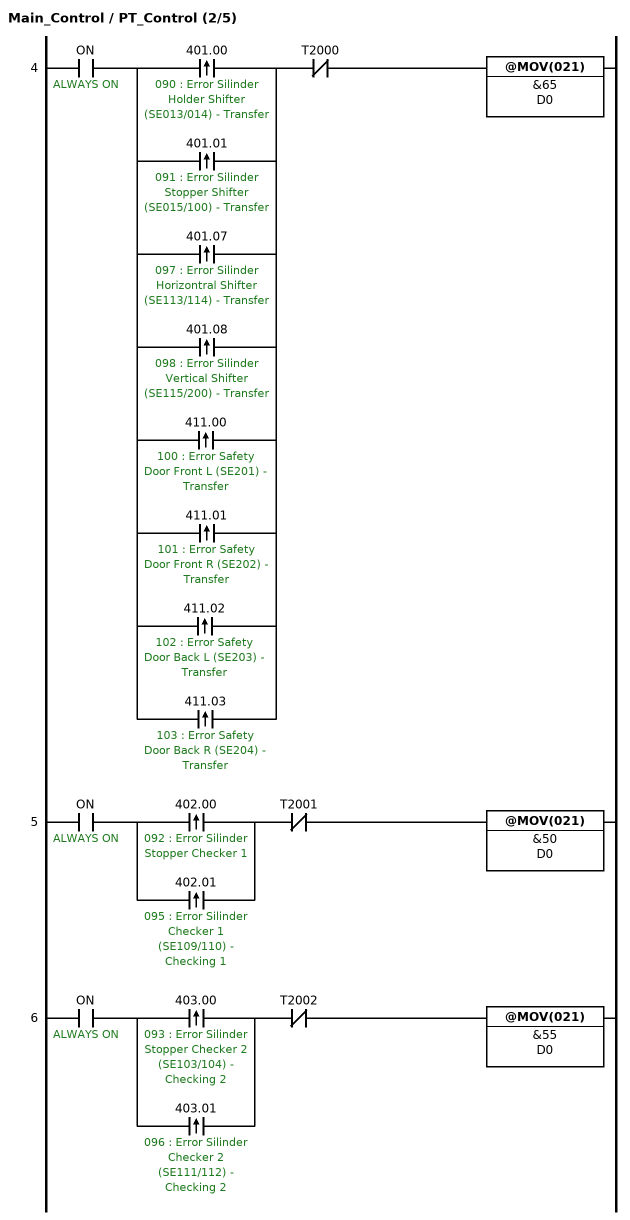
; rung 4
LD ON  ; ALWAYS ON
@LD 401.00  ; 090 : Error Silinder Holder Shifter (SE013/014) - Transfer
@OR 401.01  ; 091 : Error Silinder Stopper Shifter (SE015/100) - Transfer
@OR 401.07  ; 097 : Error Silinder Horizontral Shifter (SE113/114) - Transfer
@OR 401.08  ; 098 : Error Silinder Vertical Shifter (SE115/200) - Transfer
@OR 411.00  ; 100 : Error Safety Door Front L (SE201) - Transfer
@OR 411.01  ; 101 : Error Safety Door Front R (SE202) - Transfer
@OR 411.02  ; 102 : Error Safety Door Back L (SE203) - Transfer
@OR 411.03  ; 103 : Error Safety Door Back R (SE204) - Transfer
ANDLD
ANDNOT T2000
@MOV(021) &65 D0
; rung 5
LD ON  ; ALWAYS ON
@LD 402.00  ; 092 : Error Silinder Stopper Checker 1
@OR 402.01  ; 095 : Error Silinder Checker 1 (SE109/110) - Checking 1
ANDLD
ANDNOT T2001
@MOV(021) &50 D0
; rung 6
LD ON  ; ALWAYS ON
@LD 403.00  ; 093 : Error Silinder Stopper Checker 2 (SE103/104) - Checking 2
@OR 403.01  ; 096 : Error Silinder Checker 2 (SE111/112) - Checking 2
ANDLD
ANDNOT T2002
@MOV(021) &55 D0

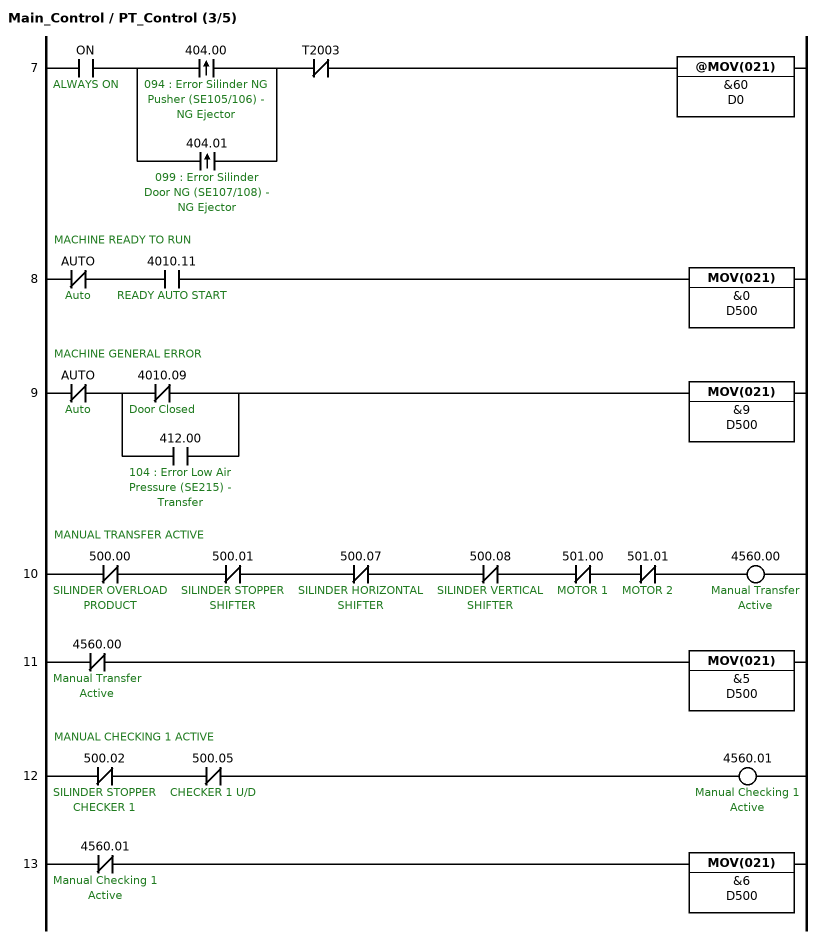
; rung 7
LD ON  ; ALWAYS ON
@LD 404.00  ; 094 : Error Silinder NG Pusher (SE105/106) - NG Ejector
@OR 404.01  ; 099 : Error Silinder Door NG (SE107/108) - NG Ejector
ANDLD
ANDNOT T2003
@MOV(021) &60 D0
; rung 8: MACHINE READY TO RUN
LDNOT AUTO  ; Auto
AND 4010.11  ; READY AUTO START
MOV(021) &0 D500
; rung 9: MACHINE GENERAL ERROR
LDNOT AUTO  ; Auto
LDNOT 4010.09  ; Door Closed
OR 412.00  ; 104 : Error Low Air Pressure (SE215) - Transfer
ANDLD
MOV(021) &9 D500
; rung 10: MANUAL TRANSFER ACTIVE
LDNOT 500.00  ; SILINDER OVERLOAD PRODUCT
ANDNOT 500.01  ; SILINDER STOPPER SHIFTER
ANDNOT 500.07  ; SILINDER HORIZONTAL SHIFTER
ANDNOT 500.08  ; SILINDER VERTICAL SHIFTER
ANDNOT 501.00  ; MOTOR 1
ANDNOT 501.01  ; MOTOR 2
OUT 4560.00  ; Manual Transfer Active
; rung 11
LDNOT 4560.00  ; Manual Transfer Active
MOV(021) &5 D500
; rung 12: MANUAL CHECKING 1 ACTIVE
LDNOT 500.02  ; SILINDER STOPPER CHECKER 1
ANDNOT 500.05  ; CHECKER 1 U/D
OUT 4560.01  ; Manual Checking 1 Active
; rung 13
LDNOT 4560.01  ; Manual Checking 1 Active
MOV(021) &6 D500

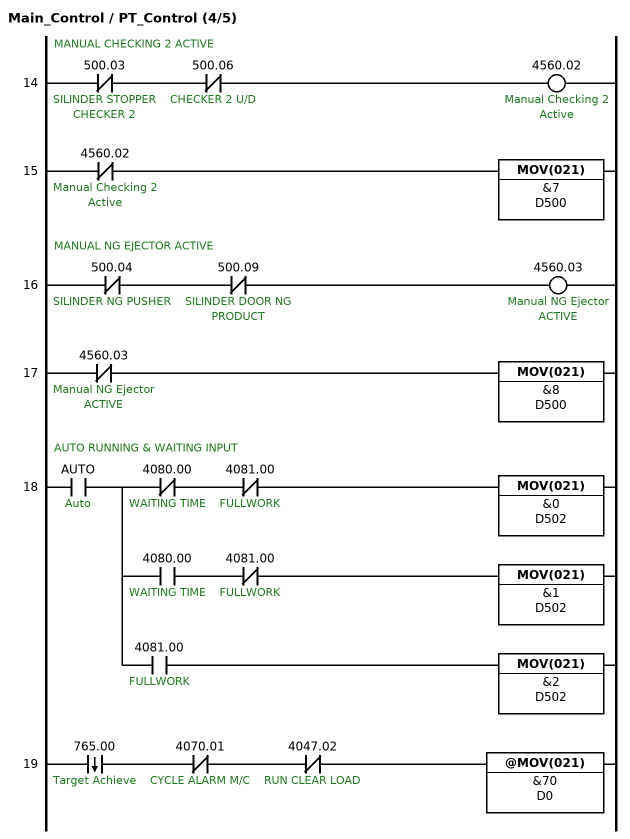
; rung 14: MANUAL CHECKING 2 ACTIVE
LDNOT 500.03  ; SILINDER STOPPER CHECKER 2
ANDNOT 500.06  ; CHECKER 2 U/D
OUT 4560.02  ; Manual Checking 2 Active
; rung 15
LDNOT 4560.02  ; Manual Checking 2 Active
MOV(021) &7 D500
; rung 16: MANUAL NG EJECTOR ACTIVE
LDNOT 500.04  ; SILINDER NG PUSHER
ANDNOT 500.09  ; SILINDER DOOR NG PRODUCT
OUT 4560.03  ; Manual NG Ejector ACTIVE
; rung 17
LDNOT 4560.03  ; Manual NG Ejector ACTIVE
MOV(021) &8 D500
; rung 18: AUTO RUNNING & WAITING INPUT
LD AUTO  ; Auto
OUT TR0
ANDNOT 4080.00  ; WAITING TIME
ANDNOT 4081.00  ; FULLWORK
MOV(021) &0 D502
LD TR0
AND 4080.00  ; WAITING TIME
ANDNOT 4081.00  ; FULLWORK
MOV(021) &1 D502
LD TR0
AND 4081.00  ; FULLWORK
MOV(021) &2 D502
; rung 19
%LD 765.00  ; Target Achieve
ANDNOT 4070.01  ; CYCLE ALARM M/C
ANDNOT 4047.02  ; RUN CLEAR LOAD
@MOV(021) &70 D0

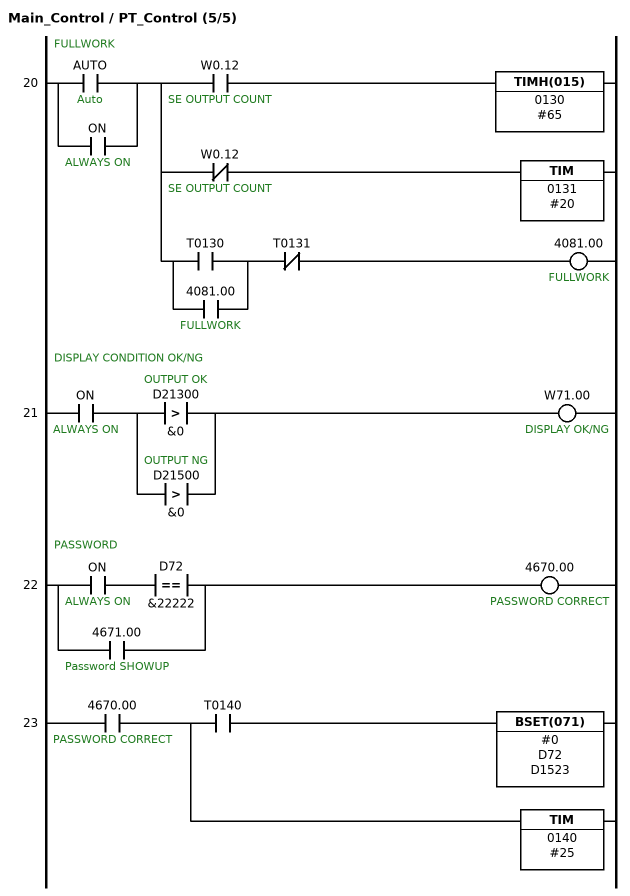
; rung 20: FULLWORK
LD AUTO  ; Auto
OR ON  ; ALWAYS ON
OUT TR0
AND W0.12  ; SE OUTPUT COUNT
TIMH(015) 0130 #65
LD TR0
ANDNOT W0.12  ; SE OUTPUT COUNT
TIM 0131 #20
LD TR0
LD T0130
OR 4081.00  ; FULLWORK
ANDLD
ANDNOT T0131
OUT 4081.00  ; FULLWORK
; rung 21: DISPLAY CONDITION OK/NG
LD ON  ; ALWAYS ON
LD>(320) D21300 &0  ; OUTPUT OK
OR>(320) D21500 &0  ; OUTPUT NG
ANDLD
OUT W71.00  ; DISPLAY OK/NG
; rung 22: PASSWORD
LD ON  ; ALWAYS ON
AND=(300) D72 &22222
OR 4671.00  ; Password SHOWUP
OUT 4670.00  ; PASSWORD CORRECT
; rung 23
LD 4670.00  ; PASSWORD CORRECT
OUT TR0
AND T0140
BSET(071) #0 D72 D1523
LD TR0
TIM 0140 #25

### Section Alarm

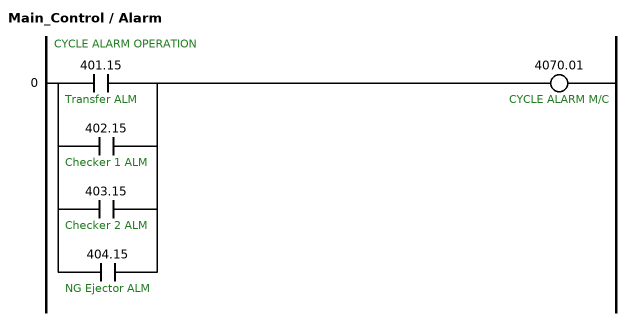
; rung 0: CYCLE ALARM OPERATION
LD 401.15  ; Transfer ALM
OR 402.15  ; Checker 1 ALM
OR 403.15  ; Checker 2 ALM
OR 404.15  ; NG Ejector ALM
OUT 4070.01  ; CYCLE ALARM M/C

### Section Record

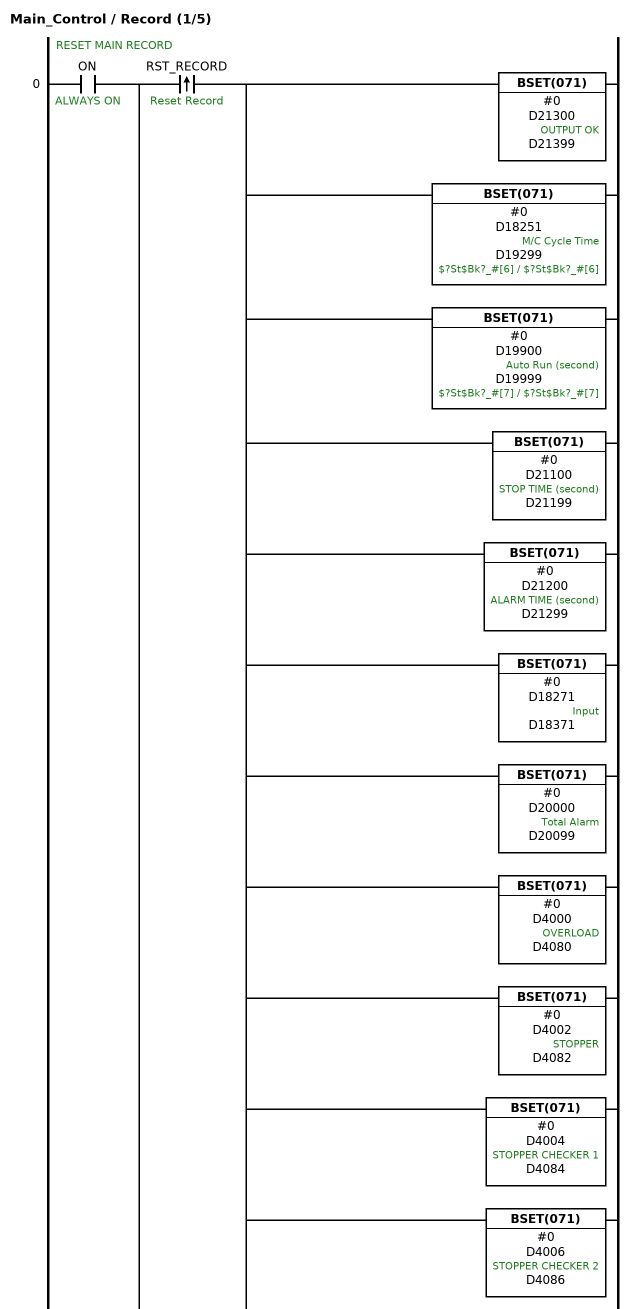

